SUBAPPLICATION PAGE (* Subapplication Type *)
  (* Standard: 61499-2 *)
  (* Version 1.0, 2023-02-07, franz *)
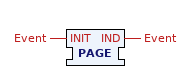
  EVENT_INPUT
    INIT;
  END_EVENT
  EVENT_OUTPUT
    IND;
  END_EVENT
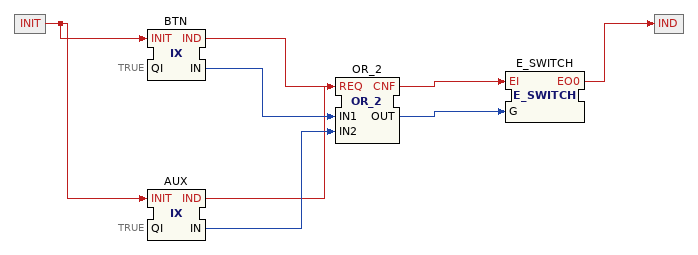
  FBS
    BTN : IX(QI := TRUE);
    AUX : IX(QI := TRUE);
    OR_2 : OR_2;
    E_SWITCH : E_SWITCH;
  END_FBS
  EVENT_CONNECTIONS
    INIT TO BTN.INIT;
    INIT TO AUX.INIT;
    BTN.IND TO OR_2.REQ;
    AUX.IND TO OR_2.REQ;
    OR_2.CNF TO E_SWITCH.EI;
    E_SWITCH.EO0 TO IND;
  END_CONNECTIONS
  DATA_CONNECTIONS
    BTN.IN TO OR_2.IN1;
    AUX.IN TO OR_2.IN2;
    OR_2.OUT TO E_SWITCH.G;
  END_CONNECTIONS
END_SUBAPPLICATION
